SUBAPPLICATION mapping_Softkeys (* Subapplication Type *)
  (* Standard: 61499-2 *)
  (* Version 1.0, 2023-01-29, Franz *)
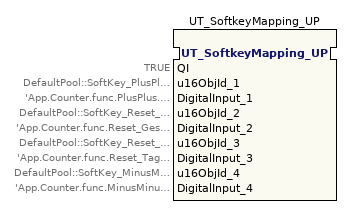
  FBS
    UT_SoftkeyMapping_UP : UT_SoftkeyMapping_UP(QI := TRUE, u16ObjId_1 := DefaultPool::SoftKey_PlusPlus, DigitalInput_1 := 'App.Counter.func.PlusPlus.SoftKey', u16ObjId_2 := DefaultPool::SoftKey_Reset_Gesamtzaehler, DigitalInput_2 := 'App.Counter.func.Reset_Gesamtzaehler.SoftKey', u16ObjId_3 := DefaultPool::SoftKey_Reset_Tageszaehler, DigitalInput_3 := 'App.Counter.func.Reset_Tageszaehler.SoftKey', u16ObjId_4 := DefaultPool::SoftKey_MinusMinus, DigitalInput_4 := 'App.Counter.func.MinusMinus.SoftKey');
  END_FBS
END_SUBAPPLICATION
